Universal Robots PolyScope program: AG_50.urp

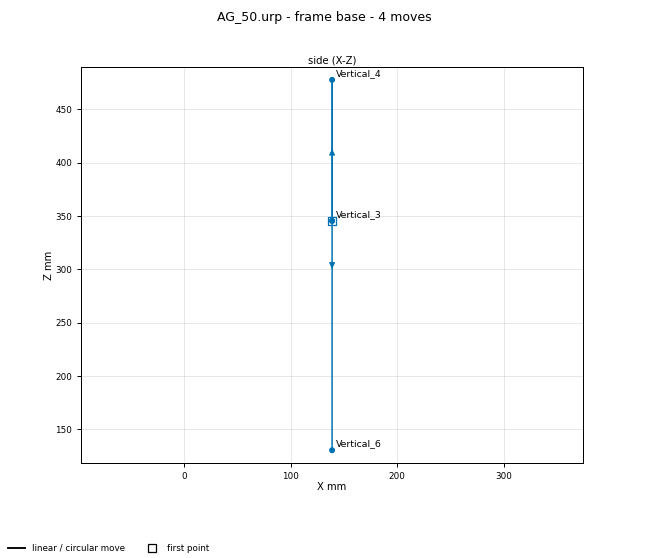
[picture p0: tool path of AG_50.urp in frame base, 4 of 4 moves have a stored position in this frame; points joined in program order, loops and branches not executed]
Program AG_50 (installation=default directory=/programs/AutoGrind createdIn=5.7.0.90932 lastSavedIn=5.11.4.108353 robotSerialNumber=20195501059)
Calibrated DH parameters: a=[0.000146, -0.418764, -0.053981, 0.000058, -0.000023, 0]; d=[0.162545, 37.319448, -206.067439, 168.881546, 0.09955, 0.099464]; alpha=[1.57004, -0.001979, 0.002304, 1.570607, -1.57066, 0]; deltaTheta=[0, -0.174616, -1.258233, 1.432844, -0.000001, 0]
Robot Program (runOnlyOnce=true)
  MoveL speed 250 mm/s, acceleration 1200 mm/s^2 (useActiveTCP=true) feature=Base
    Waypoint Vertical_3: TCP in base x=138.885 y=-597.735 z=345.466 mm, rx=0.0203 ry=0.0095 rz=0.0049 rad; joints [90.675, -74.69, 78.453, -92.586, -90.559, 180.393] deg; TCP offset x=0 y=0 z=100 mm, rx=3.1416 ry=0 rz=0 rad
    Waypoint Tilted_1: TCP in base x=138.884 y=-597.728 z=345.43 mm, rx=-0.448 ry=0.0104 rz=0.0026 rad; joints [90.791, -83.946, 99.192, -130.901, -90.87, 180.447] deg
    Waypoint Vertical_4: TCP in base x=138.908 y=-597.725 z=477.596 mm, rx=0 ry=0 rz=0.0027 rad; joints [90.516, -73.351, 57.532, -74.171, -90.073, 180.355] deg
    Waypoint Vertical_6: TCP in base x=138.876 y=-597.732 z=130.475 mm, rx=0 ry=0 rz=0.0026 rad; joints [90.482, -65.763, 99.892, -124.121, -89.984, 180.357] deg
